ABB RobotStudio station: Clasificacion.rspag

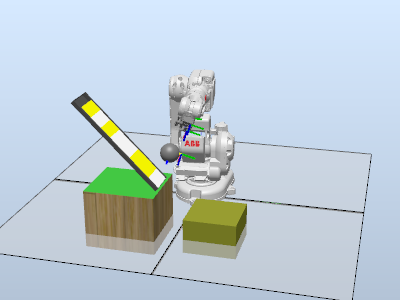
--- station ---
Station TPL2_Estacion (saved by RobotStudio 22.2.10013.1)
Controller IRB140_6_81
  mechanical unit ROB_1: IRB140_6_81_C_03, 6 joints, base frame (0, 0, 0) mm
Layout (positions relative to the parent item):
  - IRB140_6_81_C_03 [mechanism, from Robots\IRB140_6_81_C_G_03.rslib] at (0, 0, 0) mm; joint values [0.1344, 0.0114, -0.0114, -0.2281, 0.5391, 0.2641] (rad or m)
  - Mesa [part], size 365 x 405 x 340 mm
  - Deposito [part], size 300 x 300 x 200 mm
  - BloqueT1 [part] at (567.48, -115, 259.99) mm, rotated rx 45 ry 0 rz -180 deg, size 144 x 76 x 18 mm
  - BloqueT2 [part] at (567.48, -115, 259.99) mm, rotated rx 45 ry 0 rz -180 deg, size 144 x 76 x 19.5 mm
  - Slide_Base [part], size 170 x 665 x 23 mm
  - Slide_Resta [part], size 145 x 661 x 29 mm
  - Slide [part] at (567.5, -115, 260) mm, rotated rx 45 ry 0 rz 180 deg, size 174.6 x 669.2 x 29.1 mm
  - BloqueT2_2 [part] at (567.45, -114.99, 259.99) mm, rotated rx 45 ry 0 rz -180 deg, size 144 x 76 x 19.5 mm
  - BloqueT2_3 [part] at (567.46, -113.57, 261.41) mm, rotated rx 45 ry 0 rz -180 deg, size 144 x 76 x 19.5 mm
  - BloqueT2_4 [part] at (567.53, -114.99, 259.99) mm, rotated rx 45 ry 0 rz -180 deg, size 144 x 76 x 19.5 mm
  - BloqueT1_2 [part] at (567.48, -114.99, 259.99) mm, rotated rx 45 ry 0 rz -180 deg, size 144 x 76 x 18 mm
  - BloqueT1_3 [part] at (567.49, -114.99, 259.99) mm, rotated rx 45 ry 0 rz -180 deg, size 144 x 76 x 18 mm
  - BloqueT1_4 [part] at (567.49, -114.99, 259.99) mm, rotated rx 45 ry 0 rz -180 deg, size 144 x 76 x 18 mm
  - VentosayLaserRS [part] at (506.29, 60.86, 679.5) mm, rotated rx 180 ry 60 rz 180 deg, size 96.7 x 110.9 x 83.1 mm
  - Ventosa [mechanism] at (506.29, 60.86, 679.5) mm, rotated rx 180 ry 60 rz 180 deg
      TCP Ventosa at (4.41, 10.73, 83.07) mm, rotated rx 0 ry 0 rz -22.5 deg
      links: Dummy
  - FuenteLaser [mechanism] at (506.29, 60.86, 679.5) mm, rotated rx 180 ry 60 rz 180 deg
      TCP Laser at (-30.11, 31, 68.63) mm, rotated rx 0 ry 0 rz -22.5 deg
      links: Dummy
  - LaserMed [mechanism] at (506.29, 60.86, 679.5) mm, rotated rx 180 ry 60 rz 180 deg
      TCP LaserMed at (-30.11, 31, 268.63) mm, rotated rx 0 ry 0 rz -22.5 deg
      links: Dummy
  - SensorLaser [smart component]
      signals: DI SensorActivate, AO Medicion
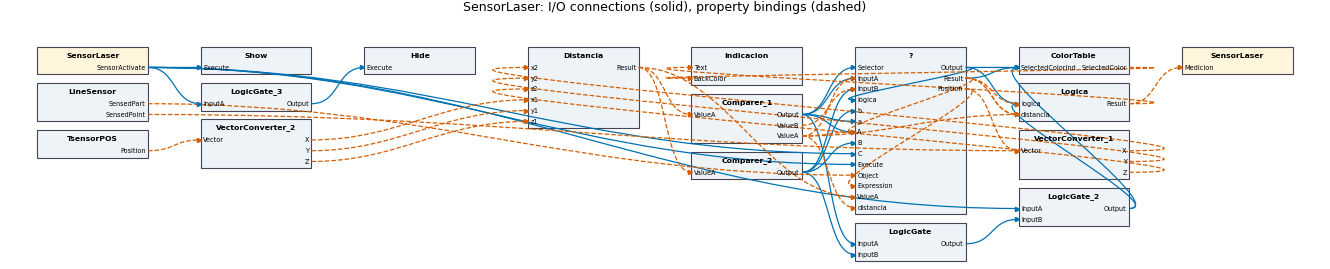
      connections:
        Comparer_1.Output -> ?.Selector
        Comparer_1.Output -> ?.InputA
        Comparer_2.Output -> ?.InputB
        ?.Output -> ?.logica
        ?.Output -> ColorTable.SelectedColorIndex
        Comparer_2.Output -> ?.b
        Comparer_1.Output -> ?.a
        ?.Output -> Logica.logica
        Comparer_1.Output -> ?.A
        Comparer_2.Output -> ?.B
        SensorLaser.SensorActivate -> ?.C
        ?.Result -> ColorTable.SelectedColorIndex
        Comparer_1.Output -> LogicGate.InputA
        Comparer_2.Output -> LogicGate.InputB
        LogicGate_2.Output -> Logica.logica
        SensorLaser.SensorActivate -> LogicGate_2.InputA
        LogicGate.Output -> LogicGate_2.InputB
        LogicGate_2.Output -> ColorTable.SelectedColorIndex
        SensorLaser.SensorActivate -> ?.Execute
        SensorLaser.SensorActivate -> Show.Execute
        LogicGate_3.Output -> Hide.Execute
        SensorLaser.SensorActivate -> LogicGate_3.InputA
        LineSensor.SensedPart => ?.Object
        ?.Position => ?.Expression
        ?.Position => VectorConverter_1.Vector
        LineSensor.SensedPoint => VectorConverter_1.Vector
        TsensorPOS.Position => VectorConverter_2.Vector
        VectorConverter_1.X => Distancia.x2
        VectorConverter_1.Y => Distancia.y2
        VectorConverter_1.Z => Distancia.z2
        VectorConverter_2.X => Distancia.x1
        VectorConverter_2.Y => Distancia.y1
        VectorConverter_2.Z => Distancia.z1
        Distancia.Result => ?.ValueA
        Distancia.Result => Comparer_1.ValueA
        Comparer_1.ValueB => ?.InputB
        Comparer_1.ValueA => ?.InputA
        Comparer_1.ValueA => ?.A
        Distancia.Result => Comparer_2.ValueA
        Logica.Result => SensorLaser.Medicion
        ?.Result => ?.A
        ?.Result => Logica.distancia
        Comparer_1.ValueA => ?.distancia
        ?.Result => Logica.logica
        ?.Result => Logica.distancia
        Comparer_1.ValueA => Logica.distancia
        Logica.Result => Indicacion.Text
        ColorTable.SelectedColor => Indicacion.BackColor
    - LineSensor [smart component, from Components\LineSensor.rslib] at (580.78, 91.86, 671.26) mm, rotated rx -146.46 ry 53.14 rz -140.36 deg
        properties: Start=[-1.11022302462516E-16 4.02455846426619E-16 0.119999533965934]; End=[-1.11022302462516E-16 4.02455846426619E-16 0.279999533965934]; Radius=0.001; SensedPart=(none); SensedPoint=[0 0 0]
      - _sensorPart_ [part], size 2 x 2 x 160 mm
    - VectorConverter_1 [smart component, from Components\VectorConverter.rslib]
        properties: X=0; Y=0; Z=0; Vector=[0 0 0]
    - TsensorPOS [smart component, from Components\PositionSensor.rslib]
        properties: Object=LineSensor; Reference=Global; ReferenceObject=(none); Position=[0.580781857400339 0.0918620590534924 0.671260890251747]; Orientation=[-2.55625298874073 0.927467979583809 -2.44975697895988]
    - VectorConverter_2 [smart component, from Components\VectorConverter.rslib]
        properties: X=0.580781857400339; Y=0.0918620590534924; Z=0.671260890251747; Vector=[0.580781857400339 0.0918620590534924 0.671260890251747]
    - Distancia [smart component, from Components\Expression.rslib]
        properties: Expression=sqrt((x2-x1)^2+(y2-y1)^2+(z2-z1)^2); Result=0.892377379005375; x2=0; x1=0.580781857400339; y2=0; y1=0.0918620590534924; z2=0; z1=0.671260890251747
    - Indicacion [smart component, from Components\MarkupControl.rslib]
        properties: Markup=Valor; Text=85; Visible=true; Position=[0.7 -0.2975 0.09]; BackColor=-65536; ForeColor=-16777216; FontSize=16; Topmost=true
    - Comparer_1 [smart component, from Components\Comparer.rslib]
        properties: ValueA=0.892377379005375; Operator=<=; ValueB=0.28
    - Comparer_2 [smart component, from Components\Comparer.rslib]
        properties: ValueA=0.892377379005375; Operator=>; ValueB=0.12
    - ColorTable [smart component, from Components\ColorTable.rslib]
        properties: NumColors=2; SelectedColorIndex=0; SelectedColor=-65536; Color0=-65536; Color1=-128
    - Logica [smart component, from Components\Expression.rslib]
        properties: Expression=OVF*(1-logica)+(200-1000*distancia)*logica; Result=85; distancia=0.892377379005375; logica=0; OVF=85
    - LogicGate [smart component, from Components\LogicGate.rslib]
        properties: Operator=AND; Delay=0
    - LogicGate_2 [smart component, from Components\LogicGate.rslib]
        properties: Operator=AND; Delay=0
    - Show [smart component, from Components\Show.rslib]
        properties: Object=LineSensor
    - LogicGate_3 [smart component, from Components\LogicGate.rslib]
        properties: Operator=NOT; Delay=0
    - Hide [smart component, from Components\Hide.rslib]
        properties: Object=LineSensor
  - EsferaTest [part] at (753.99, 31, 571.26) mm, rotated rx -146.46 ry 53.14 rz -140.36 deg, size 99.7 x 99.3 x 100 mm
Attachment: VentosayLaserRS is attached to IRB140_6_81_C_03 / Link6
Attachment: Ventosa is attached to IRB140_6_81_C_03 / Link6
Attachment: FuenteLaser is attached to IRB140_6_81_C_03 / Link6
Attachment: LaserMed is attached to IRB140_6_81_C_03 / Link6
Attachment: LineSensor is attached to FuenteLaser / Dummy
Station logic (signal -> signal, property => property):
  IRB140_6_81.DO_SON -> SensorLaser.SensorActivate
  SensorLaser.Medicion -> IRB140_6_81.AI_LS

--- Controller Data/IRB140_6_81/RAPID/TASK1/PROGMOD/LS.mod ---
MODULE LS(NOSTEPIN)
  ! VERSION 0 : primera version operativa de modulo de medicion por laser
  ! el sensor laser debe estar conectado al robot y:
  !    - la entrada analogica originalmente denominada AI10_4 renombrada como AI_LS
  !    - la salida digital originalmente denominada DO11_3 renombrada como DO_SON
  ! Módulo de control del sensor laser de distancia
  ! Este módulo permite encender, medir con distintas opciones y apagar el laser
  ! Las rutinas visibles para el usuario son:
  ! LSMeas
  !      medicion:= LSMeas(\Times:= , \TurnOff)
  !      \Times:= cantidad de veces a medir y promediar, \TurnOn \TurnOff para enceder y o apagar el sensor antes o luego de la medicion
  ! IsLSOn
  ! LSOn
  ! LSOff

  ! la entrada analógica esta mapeada y modificada desde el RAPID para entregar valores del span del sensor (-80 +80) en forma directa
  !
  ! PINOUT FICHA
  ! Ficha macho: lado sensor
  ! GND
  ! PIN 1: Ai Laser, entrada analógica de medición	: AI_LS
  ! PIN 2: DO encendido/alimentación sensor			: DO_SON
  ! PIN 3: Di entrada digital (desde sensor)		: DI_SIN
  ! PIN 4: Ai aux, desde el sensor inductivo		: AI_IS
  !
  !                   **  **
  !                ************
  !              ****************
  !             ** 4 o **** o 3 **
  !             ******************
  !             ** 2 o **** o 1 **
  !             ******************
  !                ****[==]****
  !                   ******


  ! constantes de medicion de laser
  CONST num LS_MAXVALUE:=82;
  CONST errnum ERR_LSOUTOFRNG:=77;
  LOCAL CONST num DELAY_PWR:=2;
  LOCAL CONST num DELAY_TIMES:=0.05;

  FUNC num LSMeas(
    \num Times
    \switch TurnOff)
	VAR num value:=0;
    VAR num suma:=0;
    LSOn;
    IF Present(Times) THEN
      FOR i FROM 1 TO Times DO
        suma:=suma+AI_LS;
        WaitTime DELAY_TIMES;
      ENDFOR
      value:=suma/Times;
    ELSE
      value:=AI_LS;
    ENDIF
    IF Present(TurnOff) LSOff;
    IF value>LS_MAXVALUE RAISE ERR_LSOUTOFRNG;
      !RETURN -9E+09;
      ! fuera de rango
    RETURN value;
    ERROR
        IF ERRNO=ERR_LSOUTOFRNG RAISE;
  ENDFUNC


  FUNC bool IsLSOn ()
  	IF DOutput(DO_SON)=0 THEN
  		RETURN FALSE;
  	ELSE
  		RETURN TRUE;
  	ENDIF
  ENDFUNC


  PROC LSOn() ! si el laser está ya encendido no hace nada
    IF NOT IsLSOn() THEN
    	SetDO DO_SON,1;
    	WaitTime DELAY_PWR;
    ENDIF
    ! sino no hacer nada, porque el laser ya está encendido
  ENDPROC

  PROC LSOff()
    SetDO DO_SON,0;
  ENDPROC

ENDMODULE

--- Controller Data/IRB140_6_81/RAPID/TASK1/PROGMOD/Module1.mod ---
MODULE Module1
    PERS tooldata Ventosa:=[TRUE,[[4.41,10.73,83.07],[0.980785,0,0,-0.19509]],[0.7,[0,0,45],[1,0,0,0],0,0,0]];
    PERS tooldata FuenteLaser:=[TRUE,[[-30.11,31,68.63],[0.980785,0,0,-0.19509]],[0.7,[0,0,45],[1,0,0,0],0,0,0]];
    PERS tooldata LaserMed:=[TRUE,[[-30.11,31,268.63],[0.980785,0,0,-0.19509]],[0.7,[0,0,43],[1,0,0,0],0,0,0]];
    PERS robtarget Target_10:=[[753.987,31,571.261],[0.490393,-0.168953,0.849385,-0.097545],[-1,0,-1,0],[9E+9,9E+9,9E+9,9E+9,9E+9,9E+9]];
    PERS robtarget Target_20:=[[753.987,91.8621,571.261],[0.490393,-0.168953,0.849385,-0.097545],[0,-1,0,0],[9E+9,9E+9,9E+9,9E+9,9E+9,9E+9]];
    VAR num Medicion:=0;

!***********************************************************
    !
    ! Module:  Module1
    !
    ! Description:
    !   <Insert description here>
    !
    ! Author: CARTELLI
    !
    ! Version: 1.0
    !
    !***********************************************************


    !***********************************************************
    !
    ! Procedure main
    !
    !   This is the entry point of your program
    !
    !***********************************************************
    PROC main()
        !Add your code here
        LSOn;
        Path_10;
        LSOff;
        !WaitTime 20;
    ENDPROC
    PROC Path_10()
        MoveL Target_10,v50,fine,LaserMed\WObj:=wobj0;
        Medicion:=LSMeas(\Times:=5);
        MoveL Target_20,v50,fine,LaserMed\WObj:=wobj0;
    ENDPROC
ENDMODULE

--- Controller Data/IRB140_6_81/SYSPAR/EIO.cfg ---
EIO:CFG_1.0:6:1::
#
EIO_SIGNAL:

      -Name "DO_SON" -SignalType "DO" -Access "All"

      -Name "AI_LS" -SignalType "AI" -Access "All"
